	! Debug: log final state
	Write rob_log, "";
	Write rob_log, "=== Post-move (final weld position) ===";
	cur_jt := CJointT();
	Write rob_log, "Joints: J1=" + NumToStr(cur_jt.robax.rax_1,1)
		+ " J2=" + NumToStr(cur_jt.robax.rax_2,1)
		+ " J3=" + NumToStr(cur_jt.robax.rax_3,1)
		+ " J4=" + NumToStr(cur_jt.robax.rax_4,1)
		+ " J5=" + NumToStr(cur_jt.robax.rax_5,1)
		+ " J6=" + NumToStr(cur_jt.robax.rax_6,1);
	current_tcp := CRobT(\Tool:=tWeld1\WObj:=WobjGantry);
	Write rob_log, "TCP(WobjGantry): ["
		+ NumToStr(current_tcp.trans.x,1) + ", "
		+ NumToStr(current_tcp.trans.y,1) + ", "
		+ NumToStr(current_tcp.trans.z,1) + "]";
	Write rob_log, "Orient(WobjGantry): ["
		+ NumToStr(current_tcp.rot.q1,5) + ","
		+ NumToStr(current_tcp.rot.q2,5) + ","
		+ NumToStr(current_tcp.rot.q3,5) + ","
		+ NumToStr(current_tcp.rot.q4,5) + "]";
	tcp_floor := CRobT(\Tool:=tWeld1\WObj:=WobjFloor);
	Write rob_log, "TCP(Floor): [" + NumToStr(tcp_floor.trans.x,1)
		+ "," + NumToStr(tcp_floor.trans.y,1)
		+ "," + NumToStr(tcp_floor.trans.z,1) + "]";
	TPWrite "[ROB] Post-move J1=" + NumToStr(cur_jt.robax.rax_1,1)
		+ " J4=" + NumToStr(cur_jt.robax.rax_4,1)
		+ " J5=" + NumToStr(cur_jt.robax.rax_5,1);
	TPWrite "[ROB] Final TCP (WobjGantry): ["
		+ NumToStr(current_tcp.trans.x,1) + ", "
		+ NumToStr(current_tcp.trans.y,1) + ", "
		+ NumToStr(current_tcp.trans.z,1) + "]";

	Close rob_log;

	TPWrite "========================================";
	TPWrite "[ROB] Robot move complete";
	TPWrite "========================================";
ERROR
	TPWrite "[ROB] ERROR: " + NumToStr(ERRNO,0);
	TPWrite "[ROB] Robot move failed - check configuration";
	TPWrite "========================================";
ENDPROC

! ----------------------------------------
! Generate Multi-Segment Weld Path (PlanC Phase 1)
! ----------------------------------------
! Converts start/end positions into nMotionStepCount{1} segments
! Fills pWeldPosR1{1..N} and vWeldSpeed{1..N} with linearly interpolated data
!
! Parameters:
!   adjStart/adjEnd: macro-offset-adjusted start/end positions (Floor coords)
!   refTarget: reference robtarget for robconf and extax (from CRobT)
!   nPass: current pass number (for macro torch orientation)
!
! Output: pWeldPosR1{1..nMotionStepCount{1}}, vWeldSpeed{1..nMotionStepCount{1}}
!
! Phase 1: Simple linear interpolation (calcPosStart -> calcPosEnd)
! Phase 4+: Touch sensing correction will modify positions after generation
PROC GenerateWeldPath(pos adjStart, pos adjEnd, robtarget refTarget, num nPass)
	VAR num ratio;
	VAR num i;
	VAR num nSegs;
	VAR torchmotion curMacro;

	! v1.9.55: Select buffer based on robot swap (PlanA convention)
	IF bRobSwap = FALSE THEN
		curMacro := macroStartBuffer1{nPass};
	ELSE
		curMacro := macroStartBuffer2{nPass};
	ENDIF

	nSegs := nMotionStepCount{1};
	TPWrite "[PATH] Generating " + NumToStr(nSegs,0) + " segments"
		+ " len=" + NumToStr(calcLengthWeldLine,1) + "mm"
		+ " swap=" + ValToStr(bRobSwap);

	FOR i FROM 1 TO nSegs DO
		! Linear interpolation: midpoint of each segment
		! ratio = 0.5/N for first, 1.5/N for second, ..., (N-0.5)/N for last
		ratio := (i - 0.5) / nSegs;

		! Inherit robconf and extax from current robot position
		pWeldPosR1{i} := refTarget;

		! Set interpolated position
		pWeldPosR1{i}.trans.x := adjStart.x + ratio * (adjEnd.x - adjStart.x);
		pWeldPosR1{i}.trans.y := adjStart.y + ratio * (adjEnd.y - adjStart.y);
		pWeldPosR1{i}.trans.z := adjStart.z + ratio * (adjEnd.z - adjStart.z);

		! v1.9.64: Use refTarget orientation (robot's current WobjFloor orient)
		! Fixed Floor orientations [0.5,0.5,-0.5,0.5] / [0.5,-0.5,-0.5,-0.5]
		! caused 50050 at non-zero gantry R angles (robot base rotated by R,
		! fixed Floor orient required impossible joint configs to achieve)
		! refTarget.rot is already compatible with current R angle
		! Apply torch angle adjustments (TA/WA) via RelTool on current orient
		IF bRobSwap = FALSE THEN
			pWeldPosR1{i} := RelTool(pWeldPosR1{i}, 0, 0, 0
				\Rx:=-1*curMacro.TravelAngle
				\Ry:=-1*curMacro.WorkingAngle);
		ELSE
			pWeldPosR1{i} := RelTool(pWeldPosR1{i}, 0, 0, 0
				\Rx:=curMacro.TravelAngle
				\Ry:=-1*curMacro.WorkingAngle);
		ENDIF

		! Set weld speed for this segment
		vWeldSpeed{i}.v_tcp := curMacro.WeldingSpeed;
		vWeldSpeed{i}.v_ori := 500;
		vWeldSpeed{i}.v_leax := 5000;
		vWeldSpeed{i}.v_reax := 1000;
	ENDFOR
ENDPROC

! ----------------------------------------
! BuildArcParams: Convert torchmotion buffer -> ABB arc weld data types
! v1.9.53: Maps macroStartBuffer1/macroEndBuffer1 to seam1/weld1/weave1_rob1
! v1.9.53 FIX: par4=FeedingSpeed, par6=Current (was reversed in v1.9.52)
! v1.9.53 FIX: weavedata pos5=height(0), pos6=dwellL, pos7=dir(0), pos8=dwellR
! ----------------------------------------
PROC BuildArcParams(num pass)
	VAR torchmotion curStart;
	VAR torchmotion curEnd;

	! v1.9.54: Guard - validate pass index before array access
	IF pass < 1 OR pass > MAX_WELD_PASSES THEN
		ErrWrite \W, "BuildArcParams guard", "pass=" + NumToStr(pass,0)
			+ " out of range (1-" + NumToStr(MAX_WELD_PASSES,0) + ")";
		RAISE ERR_ARGVALERR;
	ENDIF

	! v1.9.55: Select buffer based on robot swap (PlanA convention)
	IF bRobSwap = FALSE THEN
		curStart := macroStartBuffer1{pass};
		curEnd := macroEndBuffer1{pass};
	ELSE
		curStart := macroStartBuffer2{pass};
		curEnd := macroEndBuffer2{pass};
	ENDIF

	! welddata: [heat, joint_speed, heat_params{9}, cool_params{9}]
	! heat_params: [process(MIG=5), 0, voltage, wfs, 0, current, 0, 0, 0]
	! v1.9.53: par4=wfs(wire_feed_speed), par6=Current (PlanA L708)
	weld1 := [6, 0,
		[5, 0, curStart.Voltage, curStart.FeedingSpeed, 0, curStart.Current, 0, 0, 0],
		[0, 0, 0, 0, 0, 0, 0, 0, 0]];

	! seamdata: use PERS default (PlanA uses fixed seam_TRob1)
	! weld params (V/A/WFS) are in welddata, seamdata controls start/end sequence

	! weavedata: [shape, type, length, width, height, dwell_left, dir, dwell_right, 0x7]
	! v1.9.53: Fixed field positions to match ABB weavedata structure
	!          PlanA ref: Rob1_MainModule.mod L720
	!          pos5=height(0), pos6=dwell_left, pos7=dir(0), pos8=dwell_right
	weave1_rob1 := [
		curStart.WeaveShape,
		curStart.WeaveType,
		curStart.WeaveLength,
		curStart.WeaveWidth,
		0,
		curStart.WeaveDwellLeft,
		0,
		curStart.WeaveDwellRight,
		0,0,0,0,0,0,0];

	TPWrite "[ARC] Pass " + NumToStr(pass,0) + " V=" + NumToStr(curStart.Voltage,1)
		+ " WFS=" + NumToStr(curStart.FeedingSpeed,0)
		+ " A=" + NumToStr(curStart.Current,0)
		+ " swap=" + ValToStr(bRobSwap);
ENDPROC

! ----------------------------------------
! Trace Weld Line: Multi-pass weld with Approach/Retract (v2.0.0 PlanC)
! ----------------------------------------
! Moves Robot1 TCP from calcPosStart to calcPosEnd in Floor coordinates
! Uses WobjFloor for correct Floor<->World transformation
! v2.0.0 PlanC Phase 1: Multi-segment path (40-segment capable)
!
! Parameters from ConfigModule:
!   nMotionStepCount{1}: Number of active segments per pass (1-40)
!   macroStartBuffer1/macroEndBuffer1: Torch motion parameters per pass
!   nWeldPassCount: Number of active passes (1-10)
!   WELD_ARC_ENABLED: FALSE=MoveL (simulation), TRUE=ArcL (Phase 3)
!
! Flow: Approach -> MoveL(seg1) -> MoveL(seg2) -> ... -> MoveL(segN) -> Retract
PROC TraceWeldLine()
	VAR robtarget current_floor;
	VAR robtarget approach_pos;
	VAR robtarget retract_pos;
	VAR robtarget actual_floor;
	VAR pos adjStart;
	VAR pos adjEnd;
	VAR num err_x;
	VAR num err_y;
	VAR num err_z;
	VAR num err_total;
	VAR iodev trace_log;
	VAR num pass;
	VAR num seg;
	VAR num nSegs;
	VAR torchmotion curStart;
	VAR torchmotion curEnd;
	VAR robtarget pErrPos;

	TPWrite "[TRACE] TraceWeldLine v2.2.0 (PlanC Phase 1)";

	! Open own log file
	Open "HOME:/trace_weld_line.txt", trace_log \Write;
	Write trace_log, "TraceWeldLine Log (v2.0.0 PlanC) - " + CDate() + " " + CTime();
	Write trace_log, "Passes=" + NumToStr(nWeldPassCount,0)
		+ " segments=" + NumToStr(nMotionStepCount{1},0)
		+ " arc_enabled=" + ValToStr(WELD_ARC_ENABLED)
		+ " bRobSwap=" + ValToStr(bRobSwap);

	! Get current TCP in Floor coordinates (preserves robconf + extax)
	current_floor := CRobT(\Tool:=tWeld1\WObj:=WobjFloor);
	Write trace_log, "Tool=tWeld1 (design TCP)";
	Write trace_log, "Current Floor TCP=["
		+ NumToStr(current_floor.trans.x,1) + ","
		+ NumToStr(current_floor.trans.y,1) + ","
		+ NumToStr(current_floor.trans.z,1) + "]";

	nSegs := nMotionStepCount{1};

	! v1.9.54: Hard guard - reject pass count exceeding array bounds
	IF nWeldPassCount < 1 OR nWeldPassCount > MAX_WELD_PASSES THEN
		TPWrite "[TRACE] ERROR: nWeldPassCount=" + NumToStr(nWeldPassCount,0)
			+ " out of range (1-" + NumToStr(MAX_WELD_PASSES,0) + ")";
		Write trace_log, "ABORT: nWeldPassCount=" + NumToStr(nWeldPassCount,0)
			+ " exceeds MAX_WELD_PASSES=" + NumToStr(MAX_WELD_PASSES,0);
		Close trace_log;
		ErrWrite \W, "Pass count guard", "nWeldPassCount="
			+ NumToStr(nWeldPassCount,0) + " exceeds limit "
			+ NumToStr(MAX_WELD_PASSES,0);
		RAISE ERR_ARGVALERR;
	ENDIF

	! === Multi-Pass Loop ===
	FOR pass FROM 1 TO nWeldPassCount DO
		TPWrite "[TRACE] === Pass " + NumToStr(pass,0) + "/" + NumToStr(nWeldPassCount,0)
			+ " (" + NumToStr(nSegs,0) + " segments) ===";
		Write trace_log, "";
		Write trace_log, "=== Pass " + NumToStr(pass,0) + "/" + NumToStr(nWeldPassCount,0)
			+ " (" + NumToStr(nSegs,0) + " segments) ===";

		! v1.9.55: Select buffer based on robot swap (PlanA convention)
		IF bRobSwap = FALSE THEN
			curStart := macroStartBuffer1{pass};
			curEnd := macroEndBuffer1{pass};
		ELSE
			curStart := macroStartBuffer2{pass};
			curEnd := macroEndBuffer2{pass};
		ENDIF

		! --- Calculate macro-adjusted start/end positions ---
		adjStart.x := calcPosStart.x + curStart.LengthOffset;
		adjStart.z := calcPosStart.z + curStart.HeightOffset;

		adjEnd.x := calcPosEnd.x + curEnd.LengthOffset;
		adjEnd.z := calcPosEnd.z + curEnd.HeightOffset;

		! v1.9.55: BreadthOffset sign reversal on swap (PlanA convention)
		! bRobSwap=FALSE: Robot1 on A-side -> +BreadthOffset
		! bRobSwap=TRUE:  Robot1 on B-side -> -BreadthOffset (side reversed)
		IF bRobSwap = FALSE THEN
			adjStart.y := calcPosStart.y + curStart.BreadthOffset;
			adjEnd.y := calcPosEnd.y + curEnd.BreadthOffset;
		ELSE
			adjStart.y := calcPosStart.y - curStart.BreadthOffset;
			adjEnd.y := calcPosEnd.y - curEnd.BreadthOffset;
		ENDIF

		IF bRobSwap = FALSE THEN
			Write trace_log, "Buffer=Buffer1 (bRobSwap=FALSE)";
		ELSE
			Write trace_log, "Buffer=Buffer2 (bRobSwap=TRUE)";
		ENDIF
		Write trace_log, "AdjStart=[" + NumToStr(adjStart.x,1) + ","
			+ NumToStr(adjStart.y,1) + "," + NumToStr(adjStart.z,1) + "]"
			+ " TA=" + NumToStr(curStart.TravelAngle,1)
			+ " WA=" + NumToStr(curStart.WorkingAngle,1);
		Write trace_log, "AdjEnd=[" + NumToStr(adjEnd.x,1) + ","
			+ NumToStr(adjEnd.y,1) + "," + NumToStr(adjEnd.z,1) + "]"
			+ " len=" + NumToStr(calcLengthWeldLine,1) + "mm";
		Write trace_log, "Speed=" + NumToStr(curStart.WeldingSpeed,0)
			+ "mm/s V=" + NumToStr(curStart.Voltage,1)
			+ "V A=" + NumToStr(curStart.Current,0)
			+ "A WFS=" + NumToStr(curStart.FeedingSpeed,0);

		! --- Generate multi-segment path ---
		! Fills pWeldPosR1{1..nSegs} and vWeldSpeed{1..nSegs}
		GenerateWeldPath adjStart, adjEnd, current_floor, pass;
		Write trace_log, "GenerateWeldPath: " + NumToStr(nSegs,0) + " segments generated";
		! Log all generated segment positions for verification
		FOR seg FROM 1 TO nSegs DO
			Write trace_log, "  Seg " + NumToStr(seg,0)
				+ " cmd=[" + NumToStr(pWeldPosR1{seg}.trans.x,1)
				+ "," + NumToStr(pWeldPosR1{seg}.trans.y,1)
				+ "," + NumToStr(pWeldPosR1{seg}.trans.z,1) + "]"
				+ " spd=" + NumToStr(vWeldSpeed{seg}.v_tcp,0) + "mm/s";
		ENDFOR

		! --- Config check OFF for weld motion (orientation changes cause config boundary) ---
		ConfJ \Off;
		ConfL \Off;

		! --- Approach: 50mm above first segment along tool Z ---
		approach_pos := RelTool(pWeldPosR1{1}, 0, 0, -50);
		TPWrite "[TRACE] Approach (-50mm)...";
		MoveJ approach_pos, v100, fine, tWeld1 \WObj:=WobjFloor;
		Write trace_log, "Approach (-50mm) OK";

		! --- Move to first segment position ---
		TPWrite "[TRACE] MoveL to seg 1...";
		MoveL pWeldPosR1{1}, v100, fine, tWeld1 \WObj:=WobjFloor;

		! --- Verify start position ---
		actual_floor := CRobT(\Tool:=tWeld1\WObj:=WobjFloor);
		err_x := actual_floor.trans.x - pWeldPosR1{1}.trans.x;
		err_y := actual_floor.trans.y - pWeldPosR1{1}.trans.y;
		err_z := actual_floor.trans.z - pWeldPosR1{1}.trans.z;
		err_total := Sqrt(err_x*err_x + err_y*err_y + err_z*err_z);
		TPWrite "[TRACE] At seg 1 err=" + NumToStr(err_total,2) + "mm";
		Write trace_log, "Seg 1 pos=[" + NumToStr(pWeldPosR1{1}.trans.x,1) + ","
			+ NumToStr(pWeldPosR1{1}.trans.y,1) + ","
			+ NumToStr(pWeldPosR1{1}.trans.z,1) + "] err=" + NumToStr(err_total,2) + "mm";

		! --- Trace weld line: multi-segment MoveL loop ---
		IF WELD_ARC_ENABLED = TRUE THEN
			! v1.9.53: Actual ArcL welding with torchmotion -> ABB param conversion
			BuildArcParams pass;
			TPWrite "[TRACE] ARC WELD pass " + NumToStr(pass,0)
				+ " (" + NumToStr(nSegs,0) + " segs)...";
			Write trace_log, "ARC mode: V=" + NumToStr(curStart.Voltage,1)
				+ "V A=" + NumToStr(curStart.Current,0)
				+ "A WFS=" + NumToStr(curStart.FeedingSpeed,0);

			IF nSegs < 2 THEN
				! Edge case: single segment - cannot do ArcL sequence, fallback to MoveL
				TPWrite "[TRACE] WARNING: nSegs=" + NumToStr(nSegs,0) + " < 2, MoveL fallback";
				Write trace_log, "WARNING: nSegs < 2, ArcL requires min 2 segments, using MoveL";
				MoveL pWeldPosR1{1}, vWeldSpeed{1}, fine, tWeld1 \WObj:=WobjFloor;
			ELSE
				! ArcLStart: first segment (fine zone = precise arc start)
				ArcLStart pWeldPosR1{1}, vWeldSpeed{1}, seam1, weld1\Weave:=weave1_rob1,
					fine, tWeld1\WObj:=WobjFloor;
				Write trace_log, "ArcLStart seg 1 OK";

				! ArcL: intermediate segments (z1 zone = continuous path)
				FOR seg FROM 2 TO nSegs-1 DO
					ArcL pWeldPosR1{seg}, vWeldSpeed{seg}, seam1, weld1\Weave:=weave1_rob1,
						z1, tWeld1\WObj:=WobjFloor;
					Write trace_log, "ArcL seg " + NumToStr(seg,0) + " OK";
				ENDFOR

				! ArcLEnd: last segment (fine zone = precise arc end)
				ArcLEnd pWeldPosR1{nSegs}, vWeldSpeed{nSegs}, seam1, weld1\Weave:=weave1_rob1,
					fine, tWeld1\WObj:=WobjFloor;
				Write trace_log, "ArcLEnd seg " + NumToStr(nSegs,0) + " OK";
			ENDIF
		ELSE
			! Simulation: MoveL only (no arc) - with position verification
			TPWrite "[TRACE] MoveL weld pass " + NumToStr(pass,0) + " (" + NumToStr(nSegs,0) + " segs)...";
			FOR seg FROM 2 TO nSegs DO
				MoveL pWeldPosR1{seg}, vWeldSpeed{seg}, fine, tWeld1 \WObj:=WobjFloor;
				! Verify actual position after each segment (fine zone = stopped)
				actual_floor := CRobT(\Tool:=tWeld1\WObj:=WobjFloor);
				err_x := actual_floor.trans.x - pWeldPosR1{seg}.trans.x;
				err_y := actual_floor.trans.y - pWeldPosR1{seg}.trans.y;
				err_z := actual_floor.trans.z - pWeldPosR1{seg}.trans.z;
				err_total := Sqrt(err_x*err_x + err_y*err_y + err_z*err_z);
				TPWrite "[TRACE] Seg " + NumToStr(seg,0) + "/" + NumToStr(nSegs,0)
					+ " err=" + NumToStr(err_total,2) + "mm";
				Write trace_log, "Seg " + NumToStr(seg,0)
					+ " cmd=[" + NumToStr(pWeldPosR1{seg}.trans.x,1)
					+ "," + NumToStr(pWeldPosR1{seg}.trans.y,1)
					+ "," + NumToStr(pWeldPosR1{seg}.trans.z,1) + "]"
					+ " act=[" + NumToStr(actual_floor.trans.x,1)
					+ "," + NumToStr(actual_floor.trans.y,1)
					+ "," + NumToStr(actual_floor.trans.z,1) + "]"
					+ " err=" + NumToStr(err_total,2) + "mm";
			ENDFOR
		ENDIF

		! --- Final segment: MoveL to fine position ---
		MoveL pWeldPosR1{nSegs}, vWeldSpeed{nSegs}, fine, tWeld1 \WObj:=WobjFloor;

		! --- Verify end position ---
		actual_floor := CRobT(\Tool:=tWeld1\WObj:=WobjFloor);
		err_x := actual_floor.trans.x - pWeldPosR1{nSegs}.trans.x;
		err_y := actual_floor.trans.y - pWeldPosR1{nSegs}.trans.y;
		err_z := actual_floor.trans.z - pWeldPosR1{nSegs}.trans.z;
		err_total := Sqrt(err_x*err_x + err_y*err_y + err_z*err_z);
		TPWrite "[TRACE] At seg " + NumToStr(nSegs,0) + " err=" + NumToStr(err_total,2) + "mm";
		Write trace_log, "Final seg " + NumToStr(nSegs,0) + " err=" + NumToStr(err_total,2) + "mm"
			+ " dX=" + NumToStr(err_x,2) + " dY=" + NumToStr(err_y,2)
			+ " dZ=" + NumToStr(err_z,2);

		! --- Retract: 30mm above last segment along tool Z ---
		retract_pos := RelTool(pWeldPosR1{nSegs}, 0, 0, -30);
		TPWrite "[TRACE] Retract (-30mm)...";
		MoveL retract_pos, v100, fine, tWeld1 \WObj:=WobjFloor;
		Write trace_log, "Retract (-30mm) OK";

		! --- Inter-pass delay ---
		IF pass < nWeldPassCount THEN
			WaitTime 1.0;
			Write trace_log, "Inter-pass delay 1.0s";
		ENDIF
	ENDFOR

	! --- Restore config check ---
	ConfJ \On;
	ConfL \On;

	Write trace_log, "";
	Write trace_log, "TraceWeldLine complete at " + CTime();
	Close trace_log;
	TPWrite "[TRACE] TraceWeldLine complete (" + NumToStr(nWeldPassCount,0) + " passes, "
		+ NumToStr(nSegs,0) + " segs/pass)";
ERROR
	! v1.9.56: Phase 1 error handling (PlanA rArcError pattern)
	! Sequence: StopMove -> ClearPath -> StartMove -> torch retract -10mm -> Stop
	TPWrite "[TRACE] ERROR: ERRNO=" + NumToStr(ERRNO,0);
	Write trace_log, "ERROR ERRNO=" + NumToStr(ERRNO,0) + " at " + CTime();

	! Step 1: Motion safety stop - clear motion buffer
	StopMove;
	ClearPath;
	StartMove;
	TPWrite "[TRACE] StopMove->ClearPath->StartMove OK";
	Write trace_log, "StopMove->ClearPath->StartMove OK";

	! Step 2: Capture error position
	pErrPos := CRobT(\Tool:=tWeld1\WObj:=WobjFloor);
	Write trace_log, "Error pos=["
		+ NumToStr(pErrPos.trans.x,1) + ","
		+ NumToStr(pErrPos.trans.y,1) + ","
		+ NumToStr(pErrPos.trans.z,1) + "]";

	! Step 3: Torch retract -10mm along tool Z (PlanA: RelTool 0,0,-10)
	MoveL RelTool(pErrPos, 0, 0, -10), v100, z0, tWeld1\WObj:=WobjFloor;
	TPWrite "[TRACE] Torch retract -10mm OK";
	Write trace_log, "Torch retract -10mm OK";

	Write trace_log, "Phase 1 error handling complete at " + CTime();
	Close trace_log;
	Stop;
ENDPROC

! ----------------------------------------
! v1.9.57: Guard Verification (#8 TC T1~T5)
! ----------------------------------------
! Reads test values from HOME:/guard_test.txt
! Tests nWeldPassCount boundary conditions against MAX_WELD_PASSES
! Results logged to HOME:/guard_test_result.txt
PROC TestGuardVerification()
	VAR iodev cfg_file;
	VAR iodev res_file;
	VAR string line;
	VAR num nTests;
	VAR num testVal;
	VAR bool ok;
	VAR num i;
	VAR num nPass;
	VAR num nFail;

	nPass := 0;
	nFail := 0;

	TPWrite "========================================";
	TPWrite "[GUARD] Guard Verification v1.0";
	TPWrite "  MAX_WELD_PASSES=" + NumToStr(MAX_WELD_PASSES,0);
	TPWrite "========================================";

	Open "HOME:/guard_test.txt", cfg_file \Read;
	Open "HOME:/guard_test_result.txt", res_file \Write;
	Write res_file, "Guard Test Results - " + CDate() + " " + CTime();
	Write res_file, "MAX_WELD_PASSES=" + NumToStr(MAX_WELD_PASSES,0);
	Write res_file, "Version=" + TASK1_VERSION;

	! Read number of tests
	line := ReadStr(cfg_file);
	ok := StrToVal(line, nTests);

	FOR i FROM 1 TO nTests DO
		line := ReadStr(cfg_file);
		ok := StrToVal(line, testVal);

		Write res_file, "";
		Write res_file, "TC" + NumToStr(i,0) + ": nWeldPassCount=" + NumToStr(testVal,0);
		TPWrite "[GUARD] TC" + NumToStr(i,0) + " val=" + NumToStr(testVal,0);

		! Check guard condition (same logic as TraceWeldLine L4795)
		IF testVal < 1 OR testVal > MAX_WELD_PASSES THEN
			Write res_file, "  Result: REJECT (out of range)";
			Write res_file, "  Guard: " + NumToStr(testVal,0) + " not in [1,"
				+ NumToStr(MAX_WELD_PASSES,0) + "]";
			TPWrite "[GUARD] TC" + NumToStr(i,0) + " -> REJECT (expected)";
			nFail := nFail + 1;
		ELSE
			Write res_file, "  Result: PASS (in range)";
			Write res_file, "  Guard: " + NumToStr(testVal,0) + " in [1,"
				+ NumToStr(MAX_WELD_PASSES,0) + "]";
			TPWrite "[GUARD] TC" + NumToStr(i,0) + " -> PASS (expected)";
			nPass := nPass + 1;
		ENDIF
	ENDFOR

	Close cfg_file;
	Write res_file, "";
	Write res_file, "========================================";
	Write res_file, "SUMMARY: PASS=" + NumToStr(nPass,0)
		+ " REJECT=" + NumToStr(nFail,0)
		+ " TOTAL=" + NumToStr(nTests,0);
	Write res_file, "========================================";
	Close res_file;

	TPWrite "[GUARD] Complete: PASS=" + NumToStr(nPass,0)
		+ " REJECT=" + NumToStr(nFail,0);
	TPWrite "[GUARD] Results: HOME:/guard_test_result.txt";
ERROR
	TPWrite "[GUARD] ERROR: " + NumToStr(ERRNO,0);
	Close cfg_file;
	Close res_file;
ENDPROC

! ----------------------------------------
! v1.9.57: Swap Scenario Test (A~E)
! ----------------------------------------
! Reads scenario coordinates from HOME:/swap_test.txt
! Sets calcPosStart/calcPosEnd -> DefineWeldLine -> TraceWeldLine
! BreadthOffset=50mm for clear Buffer1/Buffer2 distinction
! Results logged to HOME:/swap_test_result.txt
PROC TestSwapScenarios()
	VAR iodev cfg_file;
	VAR iodev res_file;
	VAR string line;
	VAR num nScenarios;
	VAR num sx;
	VAR num sy;
	VAR num sz;
	VAR num ex;
	VAR num ey;
	VAR num ez;
	VAR bool ok;
	VAR num i;
	CONST num BREADTH_OFFSET_TEST := 50;
	VAR num adjStartY;
	VAR num adjEndY;
	VAR string bufName;
	VAR jointtarget dbg_jt;
	VAR robtarget dbg_tcp;
	VAR robtarget dbg_tcp_gantry;

	TPWrite "========================================";
	TPWrite "[SWAP] Swap Scenario Test v2.0 (motion enabled)";
	TPWrite "  BreadthOffset=" + NumToStr(BREADTH_OFFSET_TEST,0) + "mm";
	TPWrite "========================================";

	! Check linked motor sync before any gantry movement
	CheckLinkedMotorSync;

	! Set test conditions
	macroStartBuffer1{1}.BreadthOffset := BREADTH_OFFSET_TEST;
	macroEndBuffer1{1}.BreadthOffset := BREADTH_OFFSET_TEST;
	macroStartBuffer2{1}.BreadthOffset := BREADTH_OFFSET_TEST;
	macroEndBuffer2{1}.BreadthOffset := BREADTH_OFFSET_TEST;
	nWeldPassCount := 1;
	WELD_ARC_ENABLED := FALSE;

	Open "HOME:/swap_test.txt", cfg_file \Read;
	Open "HOME:/swap_test_result.txt", res_file \Write;
	Write res_file, "Swap Scenario Test Results - " + CDate() + " " + CTime();
	Write res_file, "Version=" + TASK1_VERSION;
	Write res_file, "BreadthOffset=" + NumToStr(BREADTH_OFFSET_TEST,0) + "mm";
	Write res_file, "nWeldPassCount=1, WELD_ARC_ENABLED=FALSE";

	! Read number of scenarios
	line := ReadStr(cfg_file);
	ok := StrToVal(line, nScenarios);

	FOR i FROM 1 TO nScenarios DO
		! Read 6 lines: sx, sy, sz, ex, ey, ez
		line := ReadStr(cfg_file);
		ok := StrToVal(line, sx);
		line := ReadStr(cfg_file);
		ok := StrToVal(line, sy);
		line := ReadStr(cfg_file);
		ok := StrToVal(line, sz);
		line := ReadStr(cfg_file);
		ok := StrToVal(line, ex);
		line := ReadStr(cfg_file);
		ok := StrToVal(line, ey);
		line := ReadStr(cfg_file);
		ok := StrToVal(line, ez);

		! Set weld line coordinates
		calcPosStart.x := sx;
		calcPosStart.y := sy;
		calcPosStart.z := sz;
		calcPosEnd.x := ex;
		calcPosEnd.y := ey;
		calcPosEnd.z := ez;

		Write res_file, "";
		Write res_file, "=== Scenario " + NumToStr(i,0) + "/" + NumToStr(nScenarios,0) + " ===";
		Write res_file, "Start=[" + NumToStr(sx,0) + ","
			+ NumToStr(sy,0) + "," + NumToStr(sz,0) + "]";
		Write res_file, "End=[" + NumToStr(ex,0) + ","
			+ NumToStr(ey,0) + "," + NumToStr(ez,0) + "]";
		TPWrite "[SWAP] === Scenario " + NumToStr(i,0) + "/"
			+ NumToStr(nScenarios,0) + " ===";

		! DefineWeldLine computes bRobSwap via ATan2
		DefineWeldLine;

		Write res_file, "Angle=" + NumToStr(nAngleRzStore,1) + " deg";
		Write res_file, "bRobSwap=" + ValToStr(bRobSwap);
		IF bRobSwap = FALSE THEN
			Write res_file, "Buffer=Buffer1, BreadthOffset=+"
				+ NumToStr(BREADTH_OFFSET_TEST,0) + "mm";
		ELSE
			Write res_file, "Buffer=Buffer2, BreadthOffset=-"
				+ NumToStr(BREADTH_OFFSET_TEST,0) + "mm";
		ENDIF

		TPWrite "[SWAP] Angle=" + NumToStr(nAngleRzStore,1)
			+ " bRobSwap=" + ValToStr(bRobSwap);

		! Calculation-only verification (no robot motion)
		! Replicate BreadthOffset sign logic from TraceWeldLine
		IF bRobSwap = FALSE THEN
			adjStartY := sy + BREADTH_OFFSET_TEST;
			adjEndY := ey + BREADTH_OFFSET_TEST;
			bufName := "Buffer1";
		ELSE
			adjStartY := sy - BREADTH_OFFSET_TEST;
			adjEndY := ey - BREADTH_OFFSET_TEST;
			bufName := "Buffer2";
		ENDIF

		Write res_file, "adjStart.y=" + NumToStr(adjStartY,1)
			+ " (calc.y=" + NumToStr(sy,0)
			+ " offset=" + NumToStr(adjStartY - sy,0) + ")";
		Write res_file, "adjEnd.y=" + NumToStr(adjEndY,1)
			+ " (calc.y=" + NumToStr(ey,0)
			+ " offset=" + NumToStr(adjEndY - ey,0) + ")";
		TPWrite "[SWAP] " + bufName + " adjY.offset="
			+ NumToStr(adjStartY - sy,0) + "mm";

		! v1.9.58: Motion enabled - gantry move + robot weld path
		! --- Debug: before gantry move ---
		dbg_jt := CJointT();
		Write res_file, "DBG pre-gantry: J1=" + NumToStr(dbg_jt.robax.rax_1,1)
			+ " J2=" + NumToStr(dbg_jt.robax.rax_2,1)
			+ " J3=" + NumToStr(dbg_jt.robax.rax_3,1)
			+ " J4=" + NumToStr(dbg_jt.robax.rax_4,1)
			+ " J5=" + NumToStr(dbg_jt.robax.rax_5,1)
			+ " J6=" + NumToStr(dbg_jt.robax.rax_6,1);
		Write res_file, "DBG pre-gantry: X1=" + NumToStr(dbg_jt.extax.eax_a,1)
			+ " Y=" + NumToStr(dbg_jt.extax.eax_b,1)
			+ " Z=" + NumToStr(dbg_jt.extax.eax_c,1)
			+ " R=" + NumToStr(dbg_jt.extax.eax_d,1);

		! v1.9.60: Clear interpolation objects before each scenario motion
		! Prevents 50426 "Out of interpolation objects" after multiple scenarios
		ClearPath;
		StartMove;

		TPWrite "[SWAP] Step 1: Move gantry...";
		Write res_file, "Motion: MoveGantryToWeldPosition...";
		MoveGantryToWeldPosition;

		! --- Debug: after gantry move ---
		dbg_jt := CJointT();
		dbg_tcp := CRobT(\Tool:=tWeld1\WObj:=WobjFloor);
		Write res_file, "DBG post-gantry: X1=" + NumToStr(dbg_jt.extax.eax_a,1)
			+ " Y=" + NumToStr(dbg_jt.extax.eax_b,1)
			+ " Z=" + NumToStr(dbg_jt.extax.eax_c,1)
			+ " R=" + NumToStr(dbg_jt.extax.eax_d,1);
		Write res_file, "DBG post-gantry TCP(Floor): ["
			+ NumToStr(dbg_tcp.trans.x,1) + ","
			+ NumToStr(dbg_tcp.trans.y,1) + ","
			+ NumToStr(dbg_tcp.trans.z,1) + "]";
		Write res_file, "Motion: Gantry positioned OK";

		TPWrite "[SWAP] Step 2: Move robot TCP...";
		Write res_file, "Motion: MoveRobotToWeldPosition...";
		MoveRobotToWeldPosition;

		! --- Debug: after robot move ---
		dbg_jt := CJointT();
		dbg_tcp := CRobT(\Tool:=tWeld1\WObj:=WobjFloor);
		Write res_file, "DBG post-robot: J1=" + NumToStr(dbg_jt.robax.rax_1,1)
			+ " J2=" + NumToStr(dbg_jt.robax.rax_2,1)
			+ " J3=" + NumToStr(dbg_jt.robax.rax_3,1)
			+ " J4=" + NumToStr(dbg_jt.robax.rax_4,1)
			+ " J5=" + NumToStr(dbg_jt.robax.rax_5,1)
			+ " J6=" + NumToStr(dbg_jt.robax.rax_6,1);
		Write res_file, "DBG post-robot TCP(Floor): ["
			+ NumToStr(dbg_tcp.trans.x,1) + ","
			+ NumToStr(dbg_tcp.trans.y,1) + ","
			+ NumToStr(dbg_tcp.trans.z,1) + "]";
		Write res_file, "DBG post-robot orient: ["
			+ NumToStr(dbg_tcp.rot.q1,5) + ","
			+ NumToStr(dbg_tcp.rot.q2,5) + ","
			+ NumToStr(dbg_tcp.rot.q3,5) + ","
			+ NumToStr(dbg_tcp.rot.q4,5) + "]";
		Write res_file, "Motion: Robot positioned OK";

		TPWrite "[SWAP] Step 3: TraceWeldLine (MoveL mode)...";
		Write res_file, "Motion: TraceWeldLine...";
		TraceWeldLine;
		Write res_file, "Motion: TraceWeldLine OK";

		Write res_file, "Scenario " + NumToStr(i,0) + " COMPLETE (motion OK)";
		TPWrite "[SWAP] Scenario " + NumToStr(i,0) + " DONE";

		! Return gantry to HOME between scenarios
		TPWrite "[SWAP] Returning gantry to HOME...";
		ReturnGantryToHome;

		! Return robot to init safe joints (prevent carry-over from extreme configs)
		dbg_jt := CJointT();
		dbg_jt.robax.rax_1 := 0;
		dbg_jt.robax.rax_2 := -49;
		dbg_jt.robax.rax_3 := 6;
		dbg_jt.robax.rax_4 := 0;
		dbg_jt.robax.rax_5 := 8;
		dbg_jt.robax.rax_6 := 0;
		MoveAbsJ dbg_jt, v200, fine, tWeld1;
		TPWrite "[SWAP] Robot returned to init position";

		IF i < nScenarios THEN
			WaitTime 2.0;
		ENDIF
	ENDFOR

	Close cfg_file;
	Write res_file, "";
	Write res_file, "========================================";
	Write res_file, "ALL " + NumToStr(nScenarios,0) + " SCENARIOS COMPLETE";
	Write res_file, "========================================";
	Close res_file;

	TPWrite "[SWAP] All " + NumToStr(nScenarios,0) + " scenarios complete";
	TPWrite "[SWAP] Results: HOME:/swap_test_result.txt";
ERROR
	TPWrite "[SWAP] ERROR: " + NumToStr(ERRNO,0);
	Close cfg_file;
	Close res_file;
ENDPROC

! ----------------------------------------
! Test Edge to Weld with Robot Move (v2.4.0)
! ----------------------------------------
! Combined test: Gantry positioning + Robot TCP movement
PROC TestEdgeToWeldWithRobot()
	VAR jointtarget actual_jt;
	VAR robtarget actual_tcp;

	TPWrite "========================================";
	TPWrite "[TEST] Edge to Weld + Robot Move v2.4.0";
	TPWrite "========================================";

	! Step 1: Check sync
	TPWrite "[TEST] Step 1: Check linked motor sync...";
	CheckLinkedMotorSync;

	! Step 2-3: Calculate
	TPWrite "[TEST] Step 2-3: Calculate weld position...";
	CalcCenterFromEdges;
	DefineWeldLine;

	TPWrite "[RESULT] Weld Start: [" + NumToStr(calcPosStart.x,1) + "," + NumToStr(calcPosStart.y,1) + "]";
	TPWrite "[RESULT] R-axis: " + NumToStr(nAngleRzStore,1) + " deg";

	! Step 4: Move gantry
	TPWrite "[TEST] Step 4: Move gantry...";
	MoveGantryToWeldPosition;

	actual_jt := CJointT();
	TPWrite "[VERIFY] Gantry: X=" + NumToStr(actual_jt.extax.eax_a,1)
		+ " Y=" + NumToStr(actual_jt.extax.eax_b,1)
		+ " Z=" + NumToStr(actual_jt.extax.eax_c,1)
		+ " R=" + NumToStr(actual_jt.extax.eax_d,1);

	! Step 5: Move robot
	TPWrite "[TEST] Step 5: Move robot TCP...";
	MoveRobotToWeldPosition;

	! Step 6: Verify final position
	UpdateGantryWobj;
	actual_tcp := CRobT(\Tool:=tWeld1\WObj:=WobjGantry);
	TPWrite "[VERIFY] Robot TCP tWeld1 (WobjGantry): ["
		+ NumToStr(actual_tcp.trans.x,1) + ", "
		+ NumToStr(actual_tcp.trans.y,1) + ", "
		+ NumToStr(actual_tcp.trans.z,1) + "]";

	! Step 7: Return home
	TPWrite "[TEST] Step 7: Return to HOME...";
	ReturnGantryToHome;

	TPWrite "========================================";
	TPWrite "[TEST] Edge to Weld + Robot Complete";
	TPWrite "========================================";
ENDPROC

! ----------------------------------------
! Test Full Weld Sequence with Robot2 Sync (v1.9.34)
! ----------------------------------------
! Complete weld sequence: Gantry + Robot1 + Robot2 synchronization
! Requires: TASK2 in mode 3 (Weld Sequence) or mode 9 (Test Menu with /sync)
PROC TestFullWeldSequence()
	VAR jointtarget actual_jt;
	VAR robtarget actual_tcp;
	VAR num wait_count;
	VAR num max_wait := 300;  ! 30 seconds timeout (Robot2_WeldReady may take time)
	VAR iodev logfile;

	TPWrite "========================================";
	TPWrite "[FULL] Full Weld Sequence v1.9.38";
	TPWrite "========================================";

	! Open log file
	Open "HOME:/full_weld_sequence.txt", logfile \Write;
	Write logfile, "Full Weld Sequence Log (v1.9.38) - " + CDate() + " " + CTime();
	Write logfile, "";

	! Step 0: Reset sync flags
	TPWrite "[FULL] Step 0: Reset sync flags";
	t1_weld_position_ready := FALSE;
	t1_weld_start := FALSE;
	t1_weld_done := FALSE;
	t2_weld_ready := FALSE;
	shared_bRobSwap := bRobSwap;
	Write logfile, "Sync flags reset, shared_bRobSwap=" + ValToStr(shared_bRobSwap);

	! Step 1: Check linked motor sync
	TPWrite "[FULL] Step 1: Check linked motor sync...";
	CheckLinkedMotorSync;
	Write logfile, "Step 1: Linked motor sync OK";

	! Step 2-3: Calculate weld position
	TPWrite "[FULL] Step 2-3: Calculate weld position...";
	CalcCenterFromEdges;
	DefineWeldLine;
	Write logfile, "Step 2-3: Weld Start=[" + NumToStr(calcPosStart.x,1) + "," + NumToStr(calcPosStart.y,1) + "," + NumToStr(calcPosStart.z,1) + "]";
	Write logfile, "         R-axis=" + NumToStr(nAngleRzStore,1) + " deg, bRobSwap=" + ValToStr(bRobSwap);

	! v1.9.37: Share Robot2 edge positions with TASK2
	shared_calcPosStart_r2.x := EDGE_START2_X;
	shared_calcPosStart_r2.y := EDGE_START2_Y;
	shared_calcPosStart_r2.z := EDGE_START2_Z;
	shared_calcPosEnd_r2.x := EDGE_END2_X;
	shared_calcPosEnd_r2.y := EDGE_END2_Y;
	shared_calcPosEnd_r2.z := EDGE_END2_Z;
	shared_calcLengthWeldLine := calcLengthWeldLine;
	Write logfile, "         Robot2 edge: Start=[" + NumToStr(EDGE_START2_X,0) + "," + NumToStr(EDGE_START2_Y,0) + "," + NumToStr(EDGE_START2_Z,0) + "]"
		+ " End=[" + NumToStr(EDGE_END2_X,0) + "," + NumToStr(EDGE_END2_Y,0) + "," + NumToStr(EDGE_END2_Z,0) + "]";

	TPWrite "[RESULT] Weld Start: [" + NumToStr(calcPosStart.x,1) + "," + NumToStr(calcPosStart.y,1) + "]";
	TPWrite "[RESULT] R-axis: " + NumToStr(nAngleRzStore,1) + " deg, bRobSwap=" + ValToStr(bRobSwap);

	! Step 4: Move gantry
	TPWrite "[FULL] Step 4: Move gantry...";
	MoveGantryToWeldPosition;
	actual_jt := CJointT();
	Write logfile, "Step 4: Gantry X=" + NumToStr(actual_jt.extax.eax_a,1) + " Y=" + NumToStr(actual_jt.extax.eax_b,1)
		+ " Z=" + NumToStr(actual_jt.extax.eax_c,1) + " R=" + NumToStr(actual_jt.extax.eax_d,1);

	! Step 5: Move Robot1
	TPWrite "[FULL] Step 5: Move Robot1 TCP...";
	MoveRobotToWeldPosition;
	UpdateGantryWobj;
	actual_tcp := CRobT(\Tool:=tWeld1\WObj:=WobjGantry);
	Write logfile, "Step 5: Robot1 TCP(tWeld1)=[" + NumToStr(actual_tcp.trans.x,1) + "," + NumToStr(actual_tcp.trans.y,1) + "," + NumToStr(actual_tcp.trans.z,1) + "]";

	! Step 6: Signal TASK2 (Robot2)
	TPWrite "[FULL] Step 6: Signal TASK2 (t1_weld_position_ready)...";
	t1_weld_position_ready := TRUE;
	Write logfile, "Step 6: t1_weld_position_ready=TRUE";

	! Step 7: Wait for Robot2 ready
	TPWrite "[FULL] Step 7: Waiting for Robot2 (t2_weld_ready)...";
	wait_count := 0;
	WHILE NOT t2_weld_ready DO
		WaitTime 0.1;
		wait_count := wait_count + 1;
		IF wait_count > max_wait THEN
			TPWrite "[FULL] WARNING: Robot2 timeout (continue anyway)";
			Write logfile, "Step 7: Robot2 timeout after " + NumToStr(wait_count * 0.1, 1) + "s";
			GOTO skip_r2_wait;
		ENDIF
	ENDWHILE
	TPWrite "[FULL] Robot2 ready!";
	Write logfile, "Step 7: Robot2 ready after " + NumToStr(wait_count * 0.1, 1) + "s";

skip_r2_wait:
	! Step 8: Trace weld line (multi-pass, approach/retract, RelTool orient)
	TPWrite "[FULL] Step 8: Trace weld line (" + NumToStr(nWeldPassCount,0) + " passes)...";
	Write logfile, "Step 8: TraceWeldLine start (passes=" + NumToStr(nWeldPassCount,0)
		+ " speed=" + NumToStr(macroStartBuffer1{1}.WeldingSpeed,0) + "mm/s)";
	t1_weld_start := TRUE;
	TraceWeldLine;
	Write logfile, "Step 8: TraceWeldLine complete";

	! Step 9: Signal weld done
	TPWrite "[FULL] Step 9: Signal weld done...";
	t1_weld_done := TRUE;
	WaitTime 1.0;  ! Let TASK2 process the signal
	Write logfile, "Step 9: t1_weld_done=TRUE";

	! Step 10: Reset flags and return
	TPWrite "[FULL] Step 10: Reset and return home...";
	t1_weld_position_ready := FALSE;
	t1_weld_done := FALSE;
	ReturnGantryToHome;
	Write logfile, "Step 10: Flags reset, returned home";

	! Close log
	Write logfile, "";
	Write logfile, "Full Weld Sequence completed at " + CTime();
	Close logfile;

	TPWrite "========================================";
	TPWrite "[FULL] Full Weld Sequence Complete!";
	TPWrite "========================================";
ENDPROC

! ========================================
! Command Interface (v2.1.0 - PlanA Style)
! ========================================

! ----------------------------------------
! rInit: Initialize command interface
! ----------------------------------------
PROC rInit()
	! Reset command interface
	nCmdInput := 0;
	nCmdOutput := 0;
	nCmdMatch := 0;

	! Reset motion status
	bMotionWorking := FALSE;
	bMotionFinish := TRUE;

	! Reset weld flags
	bRobSwap := FALSE;
	t1_weld_position_ready := FALSE;
	t1_weld_start := FALSE;
	t1_weld_done := FALSE;
	shared_bRobSwap := FALSE;

	TPWrite "[INIT] Command interface ready";
ENDPROC

! ----------------------------------------
! rCheckCmdMatch: Verify command acknowledgement
! ----------------------------------------
! Called after setting nCmdOutput to verify upper system received
PROC rCheckCmdMatch(num CMD)
	nCmdOutput := CMD;
	WaitUntil nCmdMatch = 1 OR nCmdMatch = -1;
	WHILE nCmdMatch <> 1 DO
		IF nCmdMatch = -1 THEN
			TPWrite "[ERROR] Command mismatch: " + NumToStr(CMD, 0);
			Stop;
		ENDIF
	ENDWHILE
	nCmdMatch := 0;
ENDPROC

! ----------------------------------------
! CommandLoop: Main command processing loop
! ----------------------------------------
! Call this from main() to enter PlanA-style command mode
PROC CommandLoop()
	VAR string sDate;
	VAR string sTime;
	VAR jointtarget abs_jt;
	VAR jointtarget inc_jt;

	TPWrite "========================================";
	TPWrite "[CMD] Entering Command Loop (v2.1.0)";
	TPWrite "[CMD] Waiting for nCmdInput...";
	TPWrite "========================================";

	WHILE TRUE DO
		! Wait for command from upper system
		WaitUntil nCmdInput <> 0;

		! Set motion status
		bMotionWorking := TRUE;
		bMotionFinish := FALSE;

		! Log timestamp and command
		sDate := CDate();
		sTime := CTime();
		sDate := StrPart(sDate, 3, 2) + StrPart(sDate, 6, 2) + StrPart(sDate, 9, 2);
		sTime := StrPart(sTime, 1, 2) + StrPart(sTime, 4, 2) + StrPart(sTime, 7, 2);
		TPWrite "[CMD] " + sDate + " " + sTime + " | Command: " + NumToStr(nCmdInput, 0);

		! Process command
		TEST nCmdInput
		CASE CMD_MOVE_TO_WORLDHOME:
			rCheckCmdMatch CMD_MOVE_TO_WORLDHOME;
			TPWrite "[CMD] Move to World Home";
			SetRobot1InitialPosition;

		CASE CMD_MOVE_ABS_GANTRY:
			rCheckCmdMatch CMD_MOVE_ABS_GANTRY;
			TPWrite "[CMD] Move Gantry Absolute";
			TPWrite "  Target: X=" + NumToStr(extGantryPos.eax_a, 1)
			       + " Y=" + NumToStr(extGantryPos.eax_b, 1)
			       + " Z=" + NumToStr(extGantryPos.eax_c, 1)
			       + " R=" + NumToStr(extGantryPos.eax_d, 1);
			abs_jt := CJointT();
			abs_jt.extax.eax_a := extGantryPos.eax_a;
			abs_jt.extax.eax_b := extGantryPos.eax_b;
			abs_jt.extax.eax_c := extGantryPos.eax_c;
			abs_jt.extax.eax_d := extGantryPos.eax_d;
			abs_jt.extax.eax_f := extGantryPos.eax_a;  ! X2 sync
			MoveAbsJ abs_jt, v500, fine, tool0;
			UpdateGantryWobj;

		CASE CMD_MOVE_INC_GANTRY:
			rCheckCmdMatch CMD_MOVE_INC_GANTRY;
			TPWrite "[CMD] Move Gantry Incremental";
			TPWrite "  Delta: X=" + NumToStr(extGantryPos.eax_a, 1)
			       + " Y=" + NumToStr(extGantryPos.eax_b, 1)
			       + " Z=" + NumToStr(extGantryPos.eax_c, 1)
			       + " R=" + NumToStr(extGantryPos.eax_d, 1);
			inc_jt := CJointT();
			inc_jt.extax.eax_a := inc_jt.extax.eax_a + extGantryPos.eax_a;
			inc_jt.extax.eax_b := inc_jt.extax.eax_b + extGantryPos.eax_b;
			inc_jt.extax.eax_c := inc_jt.extax.eax_c + extGantryPos.eax_c;
			inc_jt.extax.eax_d := inc_jt.extax.eax_d + extGantryPos.eax_d;
			inc_jt.extax.eax_f := inc_jt.extax.eax_a;  ! X2 sync
			MoveAbsJ inc_jt, v500, fine, tool0;
			UpdateGantryWobj;

		CASE CMD_WELD:
			rCheckCmdMatch CMD_WELD;
			TPWrite "[CMD] Weld (motion + arc)";
			! TODO: Implement full weld with arc
			TestWeldSequence;

		CASE CMD_WELD_MOTION:
			rCheckCmdMatch CMD_WELD_MOTION;
			TPWrite "[CMD] Weld Motion Only (no arc)";
			TestWeldSequence;

		CASE CMD_EDGE_WELD:
			rCheckCmdMatch CMD_EDGE_WELD;
			TPWrite "[CMD] Edge-based Weld";
			TestEdgeToWeld;

		CASE CMD_WIRE_CUT:
			rCheckCmdMatch CMD_WIRE_CUT;
			TPWrite "[CMD] Wire Cut (both robots)";
		CASE CMD_TEST_MENU:
			rCheckCmdMatch CMD_TEST_MENU;
			TPWrite "[CMD] Test Menu";
			TestMenu;

		CASE CMD_TEST_SINGLE:
			rCheckCmdMatch CMD_TEST_SINGLE;
			TPWrite "[CMD] Test Single Position";
			TestGantryFloorCoordinates;

		CASE CMD_TEST_ROTATION:
			rCheckCmdMatch CMD_TEST_ROTATION;
			TPWrite "[CMD] Test R-axis Rotation";
			TestGantryRotation;

		CASE CMD_TEST_MODE2:
			rCheckCmdMatch CMD_TEST_MODE2;
			TPWrite "[CMD] Test Mode2";
			TestGantryMode2;

		DEFAULT:
			TPWrite "[ERROR] Unknown command: " + NumToStr(nCmdInput, 0);
			rCheckCmdMatch 999;

		ENDTEST

		! Reset motion status
		bMotionWorking := FALSE;
		bMotionFinish := TRUE;

		! Clear command output and wait for input reset
		nCmdOutput := 0;
		WaitUntil nCmdInput = 0;

		TPWrite "[CMD] Ready for next command";
	ENDWHILE
ENDPROC

! ========================================
! ExecMoveJgJ: Execute MoveJgJ from T_Head (v1.9.61)
! ========================================
! PlanB: Move gantry + robot to target positions
! v1.9.47: Split large gantry moves into segments (ABB 50050 workaround)
! v1.9.61: FIX - Apply jRob1.robax to move robot joints (was ignored since v1.9.47)
!   MoveAbsJ is joint-space; tool0 vs tWeld1 does not affect final joint angles
PROC ExecMoveJgJ()
	VAR jointtarget jMoveTarget;
	VAR jointtarget jCurrent;
	VAR jointtarget jStep;
	VAR iodev dbg_log;
	VAR num nSegments;
	VAR num nMaxSegs;
	VAR num da;
	VAR num db;
	VAR num dc;
	VAR num dd;
	VAR num i;

	Open "HOME:/debug_movejgj.txt", dbg_log \Write;
	Write dbg_log, "ExecMoveJgJ (v1.9.61) " + CDate() + " " + CTime();

	! Read current position
	jCurrent := CJointT();
	Write dbg_log, "Current extax: a=" + NumToStr(jCurrent.extax.eax_a,1) + " b=" + NumToStr(jCurrent.extax.eax_b,1) + " c=" + NumToStr(jCurrent.extax.eax_c,1) + " d=" + NumToStr(jCurrent.extax.eax_d,1) + " f=" + NumToStr(jCurrent.extax.eax_f,1);

	! Build final target: update robot joints + gantry axes
	jMoveTarget := jCurrent;
	! v1.9.61: Apply robot joint target from T_Head
	jMoveTarget.robax := jRob1.robax;
	IF jGantry.extax.eax_a < 9E+08 THEN
		jMoveTarget.extax.eax_a := jGantry.extax.eax_a;
	ENDIF
	IF jGantry.extax.eax_b < 9E+08 THEN
		jMoveTarget.extax.eax_b := jGantry.extax.eax_b;
	ENDIF
	IF jGantry.extax.eax_c < 9E+08 THEN
		jMoveTarget.extax.eax_c := jGantry.extax.eax_c;
	ENDIF
	IF jGantry.extax.eax_d < 9E+08 THEN
		jMoveTarget.extax.eax_d := jGantry.extax.eax_d;
	ENDIF
	jMoveTarget.extax.eax_f := jMoveTarget.extax.eax_a;

	Write dbg_log, "Target extax: a=" + NumToStr(jMoveTarget.extax.eax_a,1) + " b=" + NumToStr(jMoveTarget.extax.eax_b,1) + " c=" + NumToStr(jMoveTarget.extax.eax_c,1) + " d=" + NumToStr(jMoveTarget.extax.eax_d,1) + " f=" + NumToStr(jMoveTarget.extax.eax_f,1);
	Write dbg_log, "Current robax: j1=" + NumToStr(jCurrent.robax.rax_1,1) + " j2=" + NumToStr(jCurrent.robax.rax_2,1) + " j3=" + NumToStr(jCurrent.robax.rax_3,1) + " j4=" + NumToStr(jCurrent.robax.rax_4,1) + " j5=" + NumToStr(jCurrent.robax.rax_5,1) + " j6=" + NumToStr(jCurrent.robax.rax_6,1);
	Write dbg_log, "Target robax: j1=" + NumToStr(jMoveTarget.robax.rax_1,1) + " j2=" + NumToStr(jMoveTarget.robax.rax_2,1) + " j3=" + NumToStr(jMoveTarget.robax.rax_3,1) + " j4=" + NumToStr(jMoveTarget.robax.rax_4,1) + " j5=" + NumToStr(jMoveTarget.robax.rax_5,1) + " j6=" + NumToStr(jMoveTarget.robax.rax_6,1);

	! Calculate movement per axis
	da := Abs(jMoveTarget.extax.eax_a - jCurrent.extax.eax_a);
	db := Abs(jMoveTarget.extax.eax_b - jCurrent.extax.eax_b);
	dc := Abs(jMoveTarget.extax.eax_c - jCurrent.extax.eax_c);
	dd := Abs(jMoveTarget.extax.eax_d - jCurrent.extax.eax_d);

	! Determine segments: linear max 2000mm, rotational max 45deg per segment
	nSegments := 1;
	nMaxSegs := Trunc(da / 2000) + 1;
	IF nMaxSegs > nSegments nSegments := nMaxSegs;
	nMaxSegs := Trunc(db / 2000) + 1;
	IF nMaxSegs > nSegments nSegments := nMaxSegs;
	nMaxSegs := Trunc(dc / 2000) + 1;
	IF nMaxSegs > nSegments nSegments := nMaxSegs;
	nMaxSegs := Trunc(dd / 45) + 1;
	IF nMaxSegs > nSegments nSegments := nMaxSegs;

	Write dbg_log, "Delta: a=" + NumToStr(da,0) + " b=" + NumToStr(db,0) + " c=" + NumToStr(dc,0) + " d=" + NumToStr(dd,0) + " segs=" + NumToStr(nSegments,0);
	Close dbg_log;

	IF nSegments <= 1 THEN
		! Single move - small distance
		TPWrite "[R1] MoveJgJ: single move";
		MoveAbsJ jMoveTarget, v100, fine, tool0;
	ELSE
		! Segmented move - split into steps
		TPWrite "[R1] MoveJgJ: " + NumToStr(nSegments,0) + " segments";
		FOR i FROM 1 TO nSegments DO
			jStep := jCurrent;
			! Linear interpolation for each axis
			jStep.extax.eax_a := jCurrent.extax.eax_a + (jMoveTarget.extax.eax_a - jCurrent.extax.eax_a) * i / nSegments;
			jStep.extax.eax_b := jCurrent.extax.eax_b + (jMoveTarget.extax.eax_b - jCurrent.extax.eax_b) * i / nSegments;
			jStep.extax.eax_c := jCurrent.extax.eax_c + (jMoveTarget.extax.eax_c - jCurrent.extax.eax_c) * i / nSegments;
			jStep.extax.eax_d := jCurrent.extax.eax_d + (jMoveTarget.extax.eax_d - jCurrent.extax.eax_d) * i / nSegments;
			jStep.extax.eax_f := jStep.extax.eax_a;
			! v1.9.61: Also interpolate robot joints
			jStep.robax.rax_1 := jCurrent.robax.rax_1 + (jMoveTarget.robax.rax_1 - jCurrent.robax.rax_1) * i / nSegments;
			jStep.robax.rax_2 := jCurrent.robax.rax_2 + (jMoveTarget.robax.rax_2 - jCurrent.robax.rax_2) * i / nSegments;
			jStep.robax.rax_3 := jCurrent.robax.rax_3 + (jMoveTarget.robax.rax_3 - jCurrent.robax.rax_3) * i / nSegments;
			jStep.robax.rax_4 := jCurrent.robax.rax_4 + (jMoveTarget.robax.rax_4 - jCurrent.robax.rax_4) * i / nSegments;
			jStep.robax.rax_5 := jCurrent.robax.rax_5 + (jMoveTarget.robax.rax_5 - jCurrent.robax.rax_5) * i / nSegments;
			jStep.robax.rax_6 := jCurrent.robax.rax_6 + (jMoveTarget.robax.rax_6 - jCurrent.robax.rax_6) * i / nSegments;
			IF i < nSegments THEN
				MoveAbsJ jStep, v100, z50, tool0;
			ELSE
				MoveAbsJ jStep, v100, fine, tool0;
			ENDIF
		ENDFOR
	ENDIF

	TPWrite "[R1] MoveJgJ: MoveAbsJ done";

	Open "HOME:/debug_movejgj.txt", dbg_log \Append;
	Write dbg_log, "MoveAbsJ completed (segs=" + NumToStr(nSegments,0) + ") " + CTime();
	Close dbg_log;

	UpdateGantryWobj;

	Open "HOME:/debug_movejgj.txt", dbg_log \Append;
	Write dbg_log, "UpdateGantryWobj done " + CTime();
	Write dbg_log, "ExecMoveJgJ completed OK";
	Close dbg_log;
	RETURN;

ERROR
	Open "HOME:/debug_movejgj.txt", dbg_log \Append;
	Write dbg_log, "ERROR in ExecMoveJgJ! ERRNO=" + NumToStr(ERRNO,0) + " at " + CTime();
	Close dbg_log;
	TPWrite "[R1] MoveJgJ ERROR: ERRNO=" + NumToStr(ERRNO,0);
	STOP;
ENDPROC

! ========================================
! ExecMovePgJ: Execute MovePgJ from T_Head (v1.9.41)
! ========================================
! PlanB: MoveJ to robtarget pRob1 set by T_Head
PROC ExecMovePgJ()
	MoveJ pRob1, vSync, zSync, tWeld1;
	UpdateGantryWobj;
ENDPROC

! ========================================
! ExecMovePgL: Execute MovePgL from T_Head (v1.9.41)
! ========================================
! PlanB: MoveL to robtarget pRob1 set by T_Head
PROC ExecMovePgL()
	MoveL pRob1, vSync, zSync, tWeld1;
	UpdateGantryWobj;
ENDPROC

! ========================================
! MoveAbsGantryFromExtPos: Absolute gantry move (v1.9.39)
! ========================================
! Extracted from CommandLoop CASE CMD_MOVE_ABS_GANTRY for reuse
PROC MoveAbsGantryFromExtPos()
	VAR jointtarget abs_jt;
	TPWrite "[R1] MoveAbsGantry X=" + NumToStr(extGantryPos.eax_a, 1)
	       + " Y=" + NumToStr(extGantryPos.eax_b, 1)
	       + " Z=" + NumToStr(extGantryPos.eax_c, 1)
	       + " R=" + NumToStr(extGantryPos.eax_d, 1);
	abs_jt := CJointT();
	abs_jt.extax.eax_a := extGantryPos.eax_a;
	abs_jt.extax.eax_b := extGantryPos.eax_b;
	abs_jt.extax.eax_c := extGantryPos.eax_c;
	abs_jt.extax.eax_d := extGantryPos.eax_d;
	abs_jt.extax.eax_f := extGantryPos.eax_a;  ! X2 sync
	MoveAbsJ abs_jt, v500, fine, tool0;
	UpdateGantryWobj;
ENDPROC

! ========================================
! MoveIncGantryFromExtPos: Incremental gantry move (v1.9.39)
! ========================================
! Extracted from CommandLoop CASE CMD_MOVE_INC_GANTRY for reuse
PROC MoveIncGantryFromExtPos()
	VAR jointtarget inc_jt;
	TPWrite "[R1] MoveIncGantry dX=" + NumToStr(extGantryPos.eax_a, 1)
	       + " dY=" + NumToStr(extGantryPos.eax_b, 1)
	       + " dZ=" + NumToStr(extGantryPos.eax_c, 1)
	       + " dR=" + NumToStr(extGantryPos.eax_d, 1);
	inc_jt := CJointT();
	inc_jt.extax.eax_a := inc_jt.extax.eax_a + extGantryPos.eax_a;
	inc_jt.extax.eax_b := inc_jt.extax.eax_b + extGantryPos.eax_b;
	inc_jt.extax.eax_c := inc_jt.extax.eax_c + extGantryPos.eax_c;
	inc_jt.extax.eax_d := inc_jt.extax.eax_d + extGantryPos.eax_d;
	inc_jt.extax.eax_f := inc_jt.extax.eax_a;  ! X2 sync
	MoveAbsJ inc_jt, v500, fine, tool0;
	UpdateGantryWobj;
ENDPROC

! ========================================
! rT_ROB1check: Safety position check before MoveToZHome
! ========================================
! If Robot1 is near weld line (Y<100, Z<200), move to safe Y position
PROC rT_ROB1check()
	VAR robtarget pTemp;
	pTemp := CRobT(\TaskName:="T_ROB1"\Tool:=tWeld1\WObj:=wobjWeldLine1);
	IF Abs(pTemp.trans.Y) < 100 AND Abs(pTemp.trans.Z) < 200 THEN
		IF pTemp.trans.Y > 0 THEN
			pTemp.trans.y := 130;
			MoveL pTemp, v100, fine, tWeld1\WObj:=wobjWeldLine1;
		ENDIF
		IF pTemp.trans.Y < 0 THEN
			pTemp.trans.y := -130;
			MoveL pTemp, v100, fine, tWeld1\WObj:=wobjWeldLine1;
		ENDIF
	ENDIF
ENDPROC

! ========================================
! Rob1_CommandListener: T_Head stCommand handler (v1.9.43)
! ========================================
! Responds to stCommand from T_Head task
! Protocol: "Ready" -> receive command -> execute -> "Ack" -> wait clear -> "Ready"
PROC Rob1_CommandListener()
	VAR iodev head_log;
	Open "HOME:/head_r1_listener.txt", head_log \Write;
	Write head_log, "Rob1 CommandListener (v1.9.43) - " + CDate() + " " + CTime();

	TPWrite "[R1] CommandListener started, entering Ready state";

	WHILE TRUE DO
		stReact{1} := "Ready";
		stReact{3} := "Ready";
		Write head_log, "Status: Ready, waiting stCommand...";
		WaitUntil stCommand <> "";
		Write head_log, "Received: " + stCommand;
		TPWrite "[R1] stCommand=" + stCommand;

		TEST stCommand
			CASE "MoveJgJ":
				stReact{1} := "";
				stReact{3} := "";
				ExecMoveJgJ;
				stReact{1} := "Ack";
				stReact{3} := "Ack";
				Write head_log, "MoveJgJ done";
				WaitUntil stCommand = "";

			CASE "MovePgJ":
				stReact{1} := "";
				stReact{3} := "";
				ExecMovePgJ;
				stReact{1} := "Ack";
				stReact{3} := "Ack";
				Write head_log, "MovePgJ done";
				WaitUntil stCommand = "";

			CASE "MovePgL":
				stReact{1} := "";
				stReact{3} := "";
				ExecMovePgL;
				stReact{1} := "Ack";
				stReact{3} := "Ack";
				Write head_log, "MovePgL done";
				WaitUntil stCommand = "";

			CASE "MoveHome":
				stReact{1} := "";
				stReact{3} := "";
				SetRobot1InitialPosition;
				stReact{1} := "Ack";
				stReact{3} := "Ack";
				Write head_log, "MoveHome done";
				WaitUntil stCommand = "";

			CASE "MoveMeasurementHome":
				stReact{1} := "";
				stReact{3} := "";
				! Stub - measurement home position
				stReact{1} := "Ack";
				stReact{3} := "Ack";
				Write head_log, "MoveMeasurementHome done (stub)";
				WaitUntil stCommand = "";

			CASE "MoveAbsGantry":
				stReact{1} := "";
				stReact{3} := "";
				MoveAbsGantryFromExtPos;
				stReact{1} := "Ack";
				stReact{3} := "Ack";
				Write head_log, "MoveAbsGantry done";
				WaitUntil stCommand = "";

			CASE "MoveIncGantry":
				stReact{1} := "";
				stReact{3} := "";
				MoveIncGantryFromExtPos;
				stReact{1} := "Ack";
				stReact{3} := "Ack";
				Write head_log, "MoveIncGantry done";
				WaitUntil stCommand = "";

			CASE "EdgeWeld":
				stReact{1} := "";
				stReact{3} := "";
				Write head_log, "EdgeWeld: calling TestFullWeldSequence";
				TestFullWeldSequence;
				stReact{1} := "Ack";
				stReact{3} := "Ack";
				Write head_log, "EdgeWeld done";
				WaitUntil stCommand = "";

			CASE "Weld", "WeldMotion":
				stReact{1} := "";
				stReact{3} := "";
				Write head_log, "Weld/WeldMotion: calling TestWeldSequence";
				TestWeldSequence;
				stReact{1} := "Ack";
				stReact{3} := "Ack";
				Write head_log, "Weld done";
				WaitUntil stCommand = "";

			CASE "WeldCorr", "WeldMotionCorr":
				stReact{1} := "";
				stReact{3} := "";
				Write head_log, "WeldCorr: calling TestWeldSequence (with corr)";
				TestWeldSequence;
				stReact{1} := "Ack";
				stReact{3} := "Ack";
				Write head_log, "WeldCorr done";
				WaitUntil stCommand = "";

			CASE "WireCut", "Rob1WireCut":
				stReact{1} := "";
				stReact{3} := "";
				! Stub - wire cut
				stReact{1} := "Ack";
				stReact{3} := "Ack";
				Write head_log, "WireCut done (stub)";
				WaitUntil stCommand = "";

			CASE "TestMenu":
				stReact{1} := "";
				stReact{3} := "";
				TestMenu;
				stReact{1} := "Ack";
				stReact{3} := "Ack";
				Write head_log, "TestMenu done";
				WaitUntil stCommand = "";

			CASE "TestSingle":
				stReact{1} := "";
				stReact{3} := "";
				TestGantryFloorCoordinates;
				stReact{1} := "Ack";
				stReact{3} := "Ack";
				Write head_log, "TestSingle done";
				WaitUntil stCommand = "";

			CASE "TestRotation":
				stReact{1} := "";
				stReact{3} := "";
				TestGantryRotation;
				stReact{1} := "Ack";
				stReact{3} := "Ack";
				Write head_log, "TestRotation done";
				WaitUntil stCommand = "";

			CASE "TestMode2":
				stReact{1} := "";
				stReact{3} := "";
				TestGantryMode2;
				stReact{1} := "Ack";
				stReact{3} := "Ack";
				Write head_log, "TestMode2 done";
				WaitUntil stCommand = "";

			CASE "checkpos":
				stReact{1} := "";
				stReact{3} := "";
				rT_ROB1check;
				stReact{1} := "checkposok";
				stReact{3} := "checkposok";
				Write head_log, "checkpos done";
				WaitUntil stCommand = "";

			DEFAULT:
				Write head_log, "Unknown command: " + stCommand;
				TPWrite "[R1] Unknown stCommand: " + stCommand;
				stReact{1} := "Ack";
				stReact{3} := "Ack";
				WaitUntil stCommand = "";
		ENDTEST
	ENDWHILE
ERROR
	Write head_log, "ERROR " + NumToStr(ERRNO, 0);
	Close head_log;
ENDPROC

! ============================================================
! BridgeToGantry - PlanAB-Hybrid Bridge (v0.1.0)
! ============================================================
! Copies DefineWeldLine results (calcPosStart/End, nAngleRzStore)
! into shared PERS vars (WeldsG_*) for monitoring/debug.
!
! Prerequisite: DefineWeldLine() must be called first.
! ============================================================
PROC BridgeToGantry(num weld_speed)
	WeldsG_StartX := calcPosStart.x;
	WeldsG_StartY := calcPosStart.y;
	WeldsG_StartZ := calcPosStart.z;
	WeldsG_StartR := nAngleRzStore;  ! result of DefineWeldLine()
	WeldsG_EndX   := calcPosEnd.x;
	WeldsG_EndY   := calcPosEnd.y;
	WeldsG_EndZ   := calcPosEnd.z;
	WeldsG_EndR   := nAngleRzStore;  ! same angle start=end
	WeldsG_Speed  := weld_speed;
	TPWrite "[BRIDGE] WeldsG set: Start=[" + NumToStr(WeldsG_StartX,0)
	        + "," + NumToStr(WeldsG_StartY,0) + "] End=["
	        + NumToStr(WeldsG_EndX,0) + "," + NumToStr(WeldsG_EndY,0)
	        + "] R=" + NumToStr(WeldsG_StartR,1) + "deg v=" + NumToStr(weld_speed,0);
ENDPROC

! ============================================================
! TestPlanAB_Stage1 - Hybrid Stage1 Concept Test (v0.2.0)
! ============================================================
! Reads 5 scenarios from swap_test.txt.
! Flow: DefineWeldLine -> BridgeToGantry -> MoveExtJ
! Direction-C: TASK1 drives gantry directly (no TASK7).
!
! Output: HOME:/planab_stage1.txt
! ============================================================
PROC TestPlanAB_Stage1()
	VAR iodev cfg_file;
	VAR iodev res_file;
	VAR string line;
	VAR num nScenarios;
	VAR num sx;
	VAR num sy;
	VAR num sz;
	VAR num ex;
	VAR num ey;
	VAR num ez;
	VAR bool ok;
	VAR num i;
	VAR jointtarget jt_start;
	VAR jointtarget jt_end;
	VAR pos phys;
	VAR num target_r;
	CONST num WELD_SPEED := 20;  ! mm/s

	TPWrite "========================================";
	TPWrite "[HYBRID] PlanAB Stage1 Direct MoveExtJ";
	TPWrite "Direction-C: TASK1 drives gantry directly";
	TPWrite "========================================";

	Open "HOME:/swap_test.txt", cfg_file \Read;
	Open "HOME:/planab_stage1.txt", res_file \Write;
	Write res_file, "PlanAB Hybrid Stage1 Test (Direction-C) - " + CDate() + " " + CTime();
	Write res_file, "Version=" + TASK1_VERSION;
	Write res_file, "Concept: DefineWeldLine -> BridgeToGantry -> MoveExtJ";

	! Read scenario count
	line := ReadStr(cfg_file);
	ok := StrToVal(line, nScenarios);
	IF NOT ok THEN
		TPWrite "[HYBRID] ERROR: Failed to parse scenario count";
		Write res_file, "ERROR: Failed to parse nScenarios from: " + line;
		Close cfg_file;
		Close res_file;
		RETURN;
	ENDIF
	Write res_file, "Scenarios=" + NumToStr(nScenarios,0);

	FOR i FROM 1 TO nScenarios DO
		! Read 6 lines: sx, sy, sz, ex, ey, ez
		line := ReadStr(cfg_file); ok := StrToVal(line, sx);
		line := ReadStr(cfg_file); ok := ok AND StrToVal(line, sy);
		line := ReadStr(cfg_file); ok := ok AND StrToVal(line, sz);
		line := ReadStr(cfg_file); ok := ok AND StrToVal(line, ex);
		line := ReadStr(cfg_file); ok := ok AND StrToVal(line, ey);
		line := ReadStr(cfg_file); ok := ok AND StrToVal(line, ez);
		IF NOT ok THEN
			TPWrite "[HYBRID] ERROR: Failed to parse coords in scenario " + NumToStr(i,0);
			Write res_file, "ERROR: Parse failed at Scenario " + NumToStr(i,0);
			Close cfg_file;
			Close res_file;
			RETURN;
		ENDIF

		! Set calcPosStart/End
		calcPosStart.x := sx;  calcPosStart.y := sy;  calcPosStart.z := sz;
		calcPosEnd.x   := ex;  calcPosEnd.y   := ey;  calcPosEnd.z   := ez;

		Write res_file, "";
		Write res_file, "=== Scenario " + NumToStr(i,0) + "/" + NumToStr(nScenarios,0) + " ===";
		Write res_file, "Input Start=[" + NumToStr(sx,0) + "," + NumToStr(sy,0) + "," + NumToStr(sz,0) + "]";
		Write res_file, "Input End=[" + NumToStr(ex,0) + "," + NumToStr(ey,0) + "," + NumToStr(ez,0) + "]";
		TPWrite "[HYBRID] === Scenario " + NumToStr(i,0) + "/" + NumToStr(nScenarios,0) + " ===";

		! Step 1: DefineWeldLine -> angle + swap (nAngleRzStore normalized to [-90,90])
		DefineWeldLine;
		Write res_file, "R_angle=" + NumToStr(nAngleRzStore,2) + "deg bRobSwap=" + ValToStr(bRobSwap);
		Write res_file, "Calc Start=[" + NumToStr(calcPosStart.x,0) + "," + NumToStr(calcPosStart.y,0) + "]";
		Write res_file, "Calc End=[" + NumToStr(calcPosEnd.x,0) + "," + NumToStr(calcPosEnd.y,0) + "]";

		! Step 2: BridgeToGantry -> store WeldsG_* PERS (monitoring/debug)
		BridgeToGantry WELD_SPEED;

		! Step 3: Build jointtarget using CJointT() (keeps robot joints at current pos)
		! Same pattern as MoveGantryToWeldPosition (proven working)
		! R-axis: HOME_GANTRY_R(0) - nAngleRzStore
		target_r := HOME_GANTRY_R - nAngleRzStore;

		! Start jointtarget: base = current joint pos, overwrite extax only
		jt_start := CJointT();
		phys := FloorToPhysical(calcPosStart);
		jt_start.extax.eax_a := phys.x;
		jt_start.extax.eax_b := phys.y;
		jt_start.extax.eax_c := phys.z;
		jt_start.extax.eax_d := target_r;
		jt_start.extax.eax_f := phys.x;

		! End jointtarget (same robot joints, only X/Y/Z changed)
		jt_end := jt_start;
		phys := FloorToPhysical(calcPosEnd);
		jt_end.extax.eax_a := phys.x;
		jt_end.extax.eax_b := phys.y;
		jt_end.extax.eax_c := phys.z;
		jt_end.extax.eax_f := phys.x;

		Write res_file, "Gantry Start(Phys): X=" + NumToStr(jt_start.extax.eax_a,1)
		        + " Y=" + NumToStr(jt_start.extax.eax_b,1)
		        + " R=" + NumToStr(target_r,2);
		Write res_file, "Gantry End(Phys):   X=" + NumToStr(jt_end.extax.eax_a,1)
		        + " Y=" + NumToStr(jt_end.extax.eax_b,1);

		! Step 4: Move gantry to start (MoveAbsJ: same as MoveGantryToWeldPosition)
		TPWrite "[HYBRID] Moving gantry to start...";
		MoveAbsJ jt_start, v500, fine, tool0;

		! Step 5: Move gantry to end (weld speed)
		TPWrite "[HYBRID] Weld driving...";
		MoveAbsJ jt_end, [WELD_SPEED,200,WELD_SPEED,200], fine, tool0;
		WaitRob \InPos;

		Write res_file, "Result=COMPLETE";
		TPWrite "[HYBRID] Scenario " + NumToStr(i,0) + " COMPLETE";
		WaitTime 1;
	ENDFOR

	Close cfg_file;
	Write res_file, "";
	Write res_file, "=== Test Complete ===";
	Close res_file;

	TPWrite "[HYBRID] Stage1 done. See HOME:/planab_stage1.txt";

ERROR
	TPWrite "[HYBRID] ERROR: " + NumToStr(ERRNO,0);
	Write res_file, "ERROR: " + NumToStr(ERRNO,0);
	Close cfg_file;
	Close res_file;
	TRYNEXT;
ENDPROC

ENDMODULE
